  MoveL 2056 to (223.77, 431.95, -17.53) mm, rotated rx -180 ry 0 rz -11.91 deg; joints [23.084, -21.343, 64.723, -81.917, 97.889, 133.109]
  MoveL 2057 to (223.53, 431.98, -17.53) mm, rotated rx -180 ry 0 rz -11.91 deg; joints [23.076, -21.347, 64.733, -81.921, 97.883, 133.114]
  MoveL 2058 to (223.29, 431.99, -17.53) mm, rotated rx 180 ry 0 rz -11.91 deg; joints [23.069, -21.353, 64.745, -81.925, 97.877, 133.119]
  MoveL 2059 to (223.05, 431.99, -17.52) mm, rotated rx -180 ry 0 rz -11.91 deg; joints [23.062, -21.359, 64.759, -81.929, 97.871, 133.126]
  MoveL 2060 to (-164.9, 431.99, -17.52) mm, rotated rx -180 ry 0 rz -11.91 deg; joints [11.107, -28.262, 79.844, -90.307, 89.248, 140.713]
  MoveL 2061 to (-194.97, 431.99, -17.53) mm, rotated rx 180 ry 0 rz -11.91 deg; joints [10.122, -28.555, 80.501, -91.087, 88.643, 141.084]
  MoveL 2062 to (-195.47, 431.99, -17.53) mm, rotated rx -180 ry 0 rz -11.91 deg; joints [10.106, -28.56, 80.512, -91.1, 88.633, 141.09]
  Set speed (38.1 mm/s)
  MoveL 2063 to (-196.09, 432.77, -17.53) mm, rotated rx -180 ry 0 rz -11.91 deg; joints [10.081, -28.525, 80.435, -91.119, 88.617, 141.049]
  MoveL 2064 to (-195.65, 434.72, -17.53) mm, rotated rx 180 ry 0 rz -11.91 deg; joints [10.084, -28.417, 80.2, -91.113, 88.616, 140.922]
  MoveL 2065 to (-195.51, 435.34, -16.89) mm, rotated rx 180 ry 0 rz -11.91 deg; joints [10.084, -28.412, 80.132, -91.111, 88.615, 140.859]
  Set speed (100.0 mm/s)
  MoveL 2066 to (-195.51, 435.34, 34.52) mm, rotated rx -180 ry 0 rz -11.91 deg; joints [10.073, -30.771, 80.586, -91.073, 88.572, 138.953]
  MoveL 2067 to (-195.51, 435.34, 34.52) mm, rotated rx -180 ry 0 rz -11.91 deg; joints [10.073, -30.771, 80.586, -91.073, 88.572, 138.953]
